VAR_GLOBAL
	{attribute 'pytmc' :=' pv: EM1L0:GEM:CNTRL:SP '}
	fGEM1SetpointValue : REAL:=0;
	{attribute 'pytmc' :=' pv: EM2L0:GEM:CNTRL:SP '}
	fGEM2SetpointValue : REAL:=0;
	
	
	{attribute 'pytmc' :=' pv: EM1L0:GEM:CNTRL:GO '}
	GEM1_GO : BOOL:=false;
	
	{attribute 'pytmc' :=' pv: EM2L0:GEM:CNTRL:GO '}
	GEM2_GO : BOOL:=false;
END_VAR

(* stored: Version 1.1.0.1, ProductVersion 3.1.4022.18
   GVL GVL_Control: Id {6d2a29ed-0dfc-4be1-ad02-3e5984113bf6} *)
